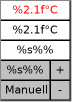
VISUALIZATION V_Heizung  // 72x102
VAR_IN_OUT
	m_Input_fbHeizregler : FB_Heizregler;
END_VAR
    Rectangle (0,60 50x20), "%s%%", text variable: m_Input_fbHeizregler.iManPHeiz, colour toggle: (m_Input_fbHeizregler.bManuell) <> 0
        OnMouseDown: write the text variable via Default
    Rectangle (0,80 50x20), "Manuell", colour toggle: (m_Input_fbHeizregler.bManuell) <> 0
        toggle m_Input_fbHeizregler.bManuell
    Rectangle (0,0 70x20), "%2.1f°C", text variable: m_Input_fbHeizregler.diTempIst * 0.01
    Rectangle (0,20 70x20), "%2.1f°C", text variable: m_Input_fbHeizregler.diTempSoll * 0.01
    Rectangle (0,40 70x20), "%s%%", text variable: m_Input_fbHeizregler.iPHeiz
        OnMouseDown: write the text variable via Edit
    Rectangle (50,60 20x20), "+", colour toggle: (m_Input_fbHeizregler.bManuell) <> 0
        OnMouseClick: execute {
            IF (m_Input_fbHeizregler.iManPHeiz < 95) THEN
            	m_Input_fbHeizregler.iManPHeiz :=
            		m_Input_fbHeizregler.iManPHeiz
            		+ 5;
            ELSE
            	m_Input_fbHeizregler.iManPHeiz := 100;
            END_IF
        }
    Rectangle (50,80 20x20), "-", colour toggle: (m_Input_fbHeizregler.bManuell) <> 0
        OnMouseClick: execute {
            IF (m_Input_fbHeizregler.iManPHeiz > 5) THEN
            	m_Input_fbHeizregler.iManPHeiz :=
            		m_Input_fbHeizregler.iManPHeiz
            		- 5;
            ELSE
            	m_Input_fbHeizregler.iManPHeiz := 0;
            END_IF
        }
END_VISUALIZATION

(* stored: Version 1.1.0.1, ProductVersion 3.1.4018.10
   Visu V_Heizung: Id {97f3489a-4654-4f32-b531-4e0917a3a6db} *)
